// TwinCAT 3 PLC project BeltSystem
// ProgramVersion: 3.1.4022.7
// libraries:
//   Tc2_Standard, * (Beckhoff Automation GmbH)
//   Tc2_System, * (Beckhoff Automation GmbH)
//   Tc3_Module, * (Beckhoff Automation GmbH)
// project tree:
//   GVLs/ GVLS.TcGVL
//   / PlcTask.TcTTO
//   POUs/ DCMOTOR.TcPOU, MAIN.TcPOU
// real-time tasks:
//   TASK PlcTask: cycle T#10ms, priority 20, ADS port 350

CONFIGURATION BeltSystem
    RESOURCE PLC ON TwinCAT3
        TASK PlcTask(INTERVAL := T#10ms, PRIORITY := 20);
        PROGRAM MAIN WITH PlcTask : MAIN;
    END_RESOURCE
END_CONFIGURATION

// ---- GVLs/GVLS.TcGVL

{attribute 'qualified_only'}
VAR_GLOBAL
//<!-- PRESPECTIVE_AUTO_INJECT_VAR_START -->
DCMotor : ARRAY [0..0] OF DCMOTOR; //Automatically Exported Collection of POU's of type 'DCMotor'
//<!-- PRESPECTIVE_AUTO_INJECT_VAR_END -->
END_VAR

// ---- POUs/MAIN.TcPOU
PROGRAM MAIN
VAR
END_VAR

END_PROGRAM

// ---- POUs/DCMOTOR.TcPOU
FUNCTION_BLOCK DCMOTOR
VAR_INPUT
//<!-- PRESPECTIVE_AUTO_INJECT_INPUT_START -->
iVelocity : REAL:= 0; //Current velocity in degrees/s
//<!-- PRESPECTIVE_AUTO_INJECT_INPUT_END -->
END_VAR
VAR_OUTPUT
//<!-- PRESPECTIVE_AUTO_INJECT_OUTPUT_START -->
oPreferredVelocity : REAL:= 0; //Preferred Velocity in degrees/s
//<!-- PRESPECTIVE_AUTO_INJECT_OUTPUT_END -->
END_VAR
VAR
//<!-- PRESPECTIVE_AUTO_INJECT_VAR_START -->
//<!-- PRESPECTIVE_AUTO_INJECT_VAR_END -->
END_VAR

END_FUNCTION_BLOCK
